{attribute 'pack_mode' := '2'} 
TYPE ST_Coordinate :
STRUCT
	fX			: LREAL;
	fY			: LREAL;
	fZ			: LREAL;
	fRx			: LREAL;
	fRy			: LREAL;
	fRz			: LREAL;
	nOriginId	: INT;
END_STRUCT
END_TYPE

(* stored: Version 1.1.0.1
   DUT ST_Coordinate: Id {21bb01c3-9903-4b8d-ab39-ac1ae75eeac2} *)
